{attribute addProperty BoxType "EK1100-0000-0018"}
{attribute addProperty Id "Beckhoff_EP2xxxEK1122Beckhoff_EP2xxxEK1122_CF43FCA125538171798695032.25"}
{attribute addProperty CRC "3002362714"}
{attribute addProperty SizeInBites "25538"}
{attribute addProperty SizeInBytes "171798695032.25"}
TYPE Beckhoff_EP2xxx_B2F46B5A EXTENDS EK1100_179A0949 :
STRUCT
	{attribute addProperty Name "Beckhoff_EP2xxxEK1122"}
	Beckhoff_EP2xxxEK1122 : Beckhoff_EP2xxxEK1122_CF43FCA1;
END_STRUCT
END_TYPE

(* stored: Version 1.2.0.0, ProductVersion 3.1.4024.9
   DUT Beckhoff_EP2xxx_B2F46B5A: Id {e946e5fa-475e-4d96-9fa7-9523052777ca} *)
